// TIA Portal V17 export
// export: Created 2023-12-05T19:31:47.8573433Z, ExportSetting WithDefaults, DisplayName Totally Integrated Automation Portal, DisplayVersion V17, DisplayName TIA Portal Openness, DisplayVersion V17, DisplayName TIA Portal Teamcenter Gateway, DisplayVersion V17, DisplayName TIA Portal Version Control Interface, DisplayVersion V17, DisplayName STEP 7 Professional, DisplayVersion V17, DisplayName STEP 7 Safety, DisplayVersion V17, DisplayName WinCC Advanced / Unified PC, DisplayVersion V17
TYPE "sPut"
// stored: IsFailsafeCompliant false
   STRUCT
      tP : Struct
         REQ : Bool;   // OUT Start sending data
         ERROR : Bool;   // OUT Error sending data
         DONE : Bool;   // OUT sending data completed successfully
         status : Int;
      END_STRUCT;
   END_STRUCT;
END_TYPE
